INTERFACE I_Room EXTENDS I_Arg

METHOD GoFault
VAR_INPUT
	sErrorText		: Str;
END_VAR
END_METHOD

METHOD GoHeat
END_METHOD

METHOD GoIdle
END_METHOD

PROPERTY Id : UDINT
GET
END_GET
END_PROPERTY

PROPERTY IsActive : BOOL
GET
END_GET
END_PROPERTY

PROPERTY IsClosed : BOOL
GET
END_GET
END_PROPERTY

PROPERTY IsOpen : BOOL
GET
END_GET
END_PROPERTY

PROPERTY IsReady : BOOL
GET
END_GET
END_PROPERTY

PROPERTY Timeout : TIME
GET
END_GET
END_PROPERTY

END_INTERFACE

(* stored: Version 1.1.0.1
   Itf I_Room: Id {988a21bf-c5a3-4b8b-8004-399623390387}
   Folder _: Id {a9fd5395-4b07-449f-a2ce-eb34a57f2518}
   Folder Flags: Id {256887b5-aed3-462f-9dfc-ed19013332c8}
   Folder Request: Id {11a83eb8-2339-4e17-8e67-0ede1cc12cb1}
   Method GoFault: Id {90bb8155-8ed3-4f0e-b5fe-88e6a4db01e4}
   Method GoHeat: Id {95c828ce-643d-497e-a695-1a3e9ecabc01}
   Method GoIdle: Id {6c54e25f-ff82-45a7-bb7f-9ff8e13440f1}
   Property Id: Id {b1b6dbeb-3191-4415-bdd6-aaa43aa69f14}
   Get Get: Id {e1adc6c7-bb71-4dca-8b9d-869d36562259}
   Property IsActive: Id {a3a76c51-bc11-490c-bc08-0e8b504978bb}
   Get Get: Id {efd159a6-0b6c-40c8-aee0-c60f42255b76}
   Property IsClosed: Id {76fbbae7-a8c5-4f9e-a5df-23b12afedadf}
   Get Get: Id {ad0db52b-1b7a-4a07-bff4-b9f152e2e91f}
   Property IsOpen: Id {d385eabe-3a2b-4540-9831-c0025bed6028}
   Get Get: Id {de7bc9b7-9fdb-4a24-b8fb-4bd11a89ab07}
   Property IsReady: Id {80f15f07-bb29-45e4-9810-30157d256069}
   Get Get: Id {c3245dfb-f3e0-4831-9299-e78a17d8a441}
   Property Timeout: Id {df00084c-cbe1-4c7d-ae4a-aca9bb4c4a87}
   Get Get: Id {f422d9e1-9cff-4591-94af-1911ba9f57f6} *)
